// TIA Portal V20 export
TYPE "typeCmHmiInterfaceSoftCam"
// stored: Access Published, Namespace Unit1.Em5
   STRUCT
      transferPnPLeftAxisX : "Unit1.Em5.typeCmHmiInterfaceSoftCamtransferPnPLeftAxisX";
      transferPnPLeftAxisY : "Unit1.Em5.typeCmHmiInterfaceSoftCamtransferPnPLeftAxisY";
      transferPnPLeftAxisZ : "Unit1.Em5.typeCmHmiInterfaceSoftCamtransferPnPLeftAxisZ";
      transferPnPRightAxisX : "Unit1.Em5.typeCmHmiInterfaceSoftCamtransferPnPRightAxisX";
      transferPnPRightAxisY : "Unit1.Em5.typeCmHmiInterfaceSoftCamtransferPnPRightAxisY";
      transferPnPRightAxisZ : "Unit1.Em5.typeCmHmiInterfaceSoftCamtransferPnPRightAxisZ";
   END_STRUCT;
END_TYPE
